(* Schneider Machine Expert - Basic project Questao3.8_FelipeV1_20241014, file version 2.9.0.0 *)
(* ProjectInformations: Name=Novo projeto *)

HARDWARE
  Cpu 0: TM221M16R/G
  EthernetConfiguration: NetworkName=M221, IpAllocationMode=FixedAddress, IpAddress=0.0.0.0, SubnetMask=0.0.0.0
  SerialLineConfiguration: Baud=Baud19200, Parity=ParityEven, DataBits=DataBits8, StopBits=StopBits1, PhysicalMedium=PhysicalMediumRs485, TransmissionMode=TransmissionModeModbusRtu, SlaveId=1, Addressing=SlaveAddressing
  MastTask: UsePeriodScanMode=false, PeriodScan=100
  FastTask: Period=255
  CpuBehavior: StartingMode=StartAsPreviousState, AutoSaveRamOnEeprom=true, WatchdogPeriod=250

SYMBOLS  (address, symbol, comment, settings)
  %M0       BOTAO
  %M1       LIGA_SENS
  %M10      LIGA_ESTEI
  %M11      DESL_ESTEI
  %M12      ATUA_SENSOR_OPTI
  %TM0        [Preset=5, Base=OneSecond]
  %I0.0     BOT_LIGA
  %I0.1     BOT_SENS
  %Q0.1     ATUA_ESTEI
  %Q0.2     DESA_ESTEI

POU Entrada
  (* SectionNumber=1 *)

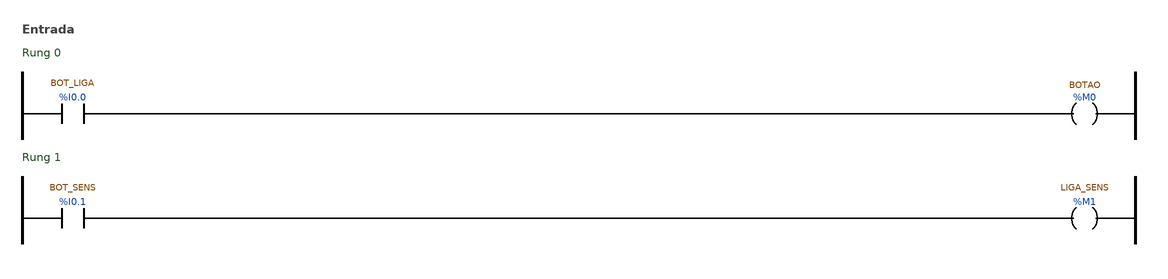

// Rung 0
  LD %I0.0                (* BOT_LIGA *)
  ST %M0                  (* BOTAO *)
  // as ST:
  //   BOTAO := BOT_LIGA;

// Rung 1
  LD %I0.1                (* BOT_SENS *)
  ST %M1                  (* LIGA_SENS *)
  // as ST:
  //   LIGA_SENS := BOT_SENS;

POU Lógica
  (* SectionNumber=2 *)

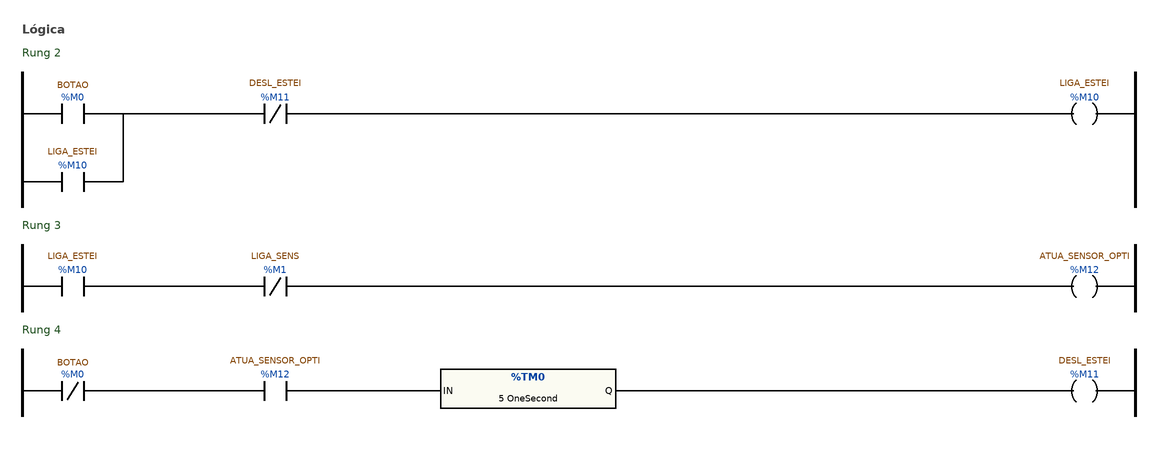

// Rung 2
  LD %M0                  (* BOTAO *)
  OR %M10                 (* LIGA_ESTEI *)
  ANDN %M11               (* DESL_ESTEI *)
  ST %M10                 (* LIGA_ESTEI *)
  // as ST:
  //   LIGA_ESTEI := (BOTAO OR LIGA_ESTEI) AND NOT DESL_ESTEI;

// Rung 3
  LD %M10                 (* LIGA_ESTEI *)
  ANDN %M1                (* LIGA_SENS *)
  ST %M12                 (* ATUA_SENSOR_OPTI *)
  // as ST:
  //   ATUA_SENSOR_OPTI := LIGA_ESTEI AND NOT LIGA_SENS;

// Rung 4
  BLK %TM0
  LDN %M0                 (* BOTAO *)
  AND %M12                (* ATUA_SENSOR_OPTI *)
  IN
  OUT_BLK
  LD Q
  ST %M11                 (* DESL_ESTEI *)
  END_BLK
  // as ST:
  //   %TM0(IN := NOT BOTAO AND ATUA_SENSOR_OPTI);
  //   DESL_ESTEI := %TM0.Q;

POU Saída
  (* SectionNumber=3 *)

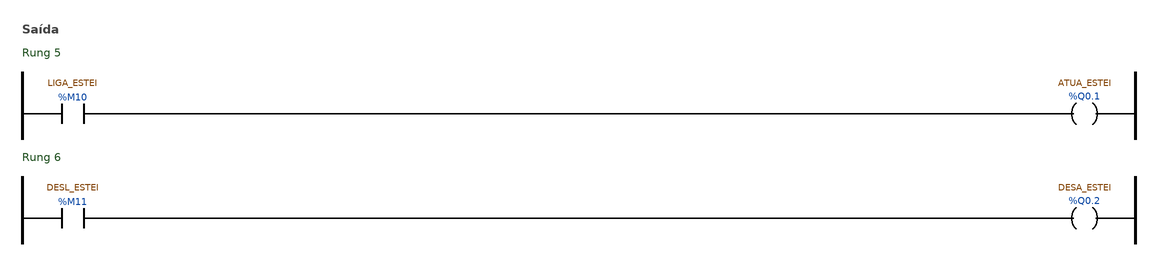

// Rung 5
  LD %M10                 (* LIGA_ESTEI *)
  ST %Q0.1                (* ATUA_ESTEI *)
  // as ST:
  //   ATUA_ESTEI := LIGA_ESTEI;

// Rung 6
  LD %M11                 (* DESL_ESTEI *)
  ST %Q0.2                (* DESA_ESTEI *)
  // as ST:
  //   DESA_ESTEI := DESL_ESTEI;
